# EPICS autosave request: IOCs/MS_DAQ/MSApp/Db/MS_TwoThetaStep_settings.req
# This file is used by autosave to determine what PVs to save (currently, autosave not used)
# It is also used by MS DAQ to determine what PVs to create

# This file contains all of the PVs used by the twoThetaStep class.

$(P)UseRobot

####################
# Diffractometer Control
####################

$(P)$(R)TwoThetaMotorName
$(P)$(R)SpinnerMotorName

####################
# Sample Container Control
##################

$(P)$(R)SCMotorName
